FUNCTION_BLOCK FB_BWK_Input
VAR_INPUT
	IN_Leistung			: SINT;	(* 0..100 % *)
	IN_Temp_Ist			: REAL;
END_VAR
VAR_OUTPUT
	Leistung				: SINT;	(* 0..100 % *)
	Temp_Ist			: REAL;
END_VAR
VAR
END_VAR

IN_Leistung		:= Leistung;
IN_Temp_Ist		:= Temp_Ist;

END_FUNCTION_BLOCK

(* stored: Version 1.1.0.1, ProductVersion 3.1.4024.9
   POU FB_BWK_Input: Id {2749fb2b-8e5d-4df6-aa41-efe656e59158}, SpecialFunc None *)
